FUNCTION_BLOCK Plant
  (* Standard: 61499-2 *)
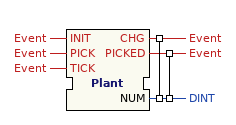
  EVENT_INPUT
    INIT;
    PICK;
    TICK;
  END_EVENT
  EVENT_OUTPUT
    CHG WITH NUM;
    PICKED WITH NUM;
  END_EVENT
  VAR_OUTPUT
    NUM : DINT;
  END_VAR
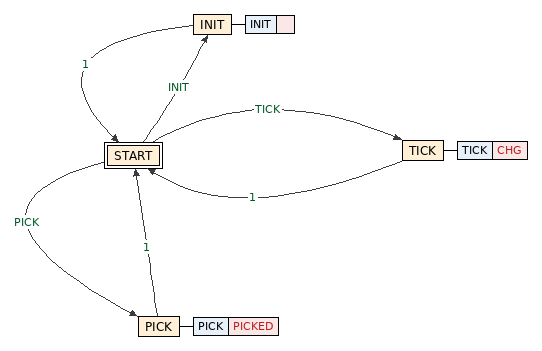
  EC_STATES
    START;
    INIT : INIT;
    TICK : TICK -> CHG;
    PICK : PICK -> PICKED;
  END_STATES
  EC_TRANSITIONS
    START TO INIT := INIT;
    INIT TO START := 1;
    START TO TICK := TICK;
    TICK TO START := 1;
    START TO PICK := PICK;
    PICK TO START := 1;
  END_TRANSITIONS
  ALGORITHM INIT IN ST:
current := 0;&#10;
  END_ALGORITHM
  ALGORITHM TICK IN ST:
current := (current + 1) MOD 10;&#10;NUM := current;&#10;
  END_ALGORITHM
  ALGORITHM PICK IN ST:
NUM := current;&#10;
  END_ALGORITHM
END_FUNCTION_BLOCK
